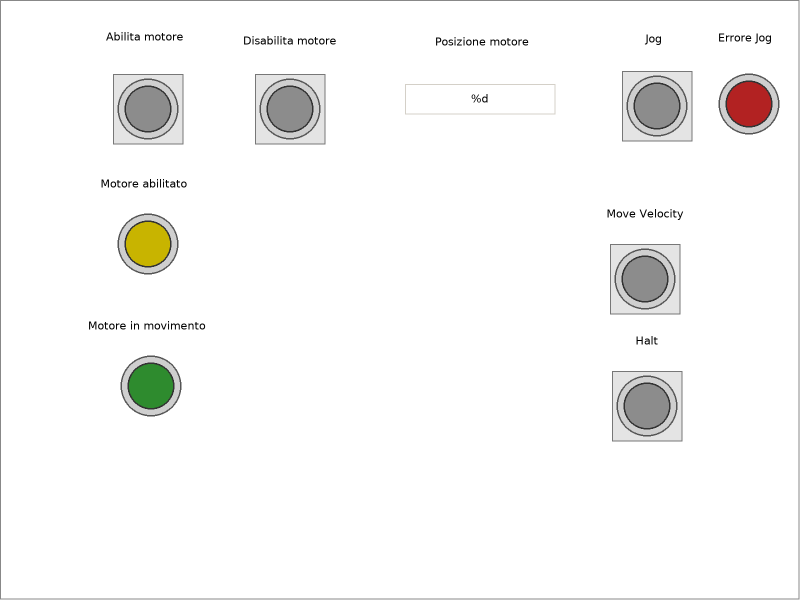
VISUALIZATION Visualization  // 800x600
    PushSwitch (113,74 70x70), variable: GVL.pAbilitaMotore, behaviour: TAP, style: Switch-PushSwitch-Gray
    Lamp1 (113,209 70x70), variable: GVL.motoreAbilitato, style: Lamp-Lamp1-Yellow
    Label (69,169 150x30), "Motore abilitato"
    Label (70,22 150x30), "Abilita motore"
    PushSwitch (255,74 70x70), variable: GVL.pDisabilitaMotore, behaviour: TAP, style: Switch-PushSwitch-Gray
    Label (215,26 150x30), "Disabilita motore"
    Textfield (405,84 150x30), "%d", text variable: GVL.Axis.NcToPlc.ActPos
    PushSwitch (622,71 70x70), variable: GVL.pAbilitaJog, behaviour: TAP, style: Switch-PushSwitch-Gray
    Label (579,24 150x30), "Jog"
    Lamp1 (116,351 70x70), variable: GVL.Axis.Status.Moving, style: Lamp-Lamp1-Green
    Label (72,311 150x30), "Motore in movimento"
    Lamp1 (714,69 70x70), variable: GVL.bErrorJog, style: Lamp-Lamp1-Red
    Label (670,23 150x30), "Errore Jog"
    Label (407,27 150x30), "Posizione motore"
    PushSwitch (610,244 70x70), variable: GVL.pMoveVelocity, behaviour: TAP, style: Switch-PushSwitch-Gray
    Label (570,199 150x30), "Move Velocity"
    PushSwitch (612,371 70x70), variable: GVL.pHalt, behaviour: TAP, style: Switch-PushSwitch-Gray
    Label (572,326 150x30), "Halt"
END_VISUALIZATION

(* stored: Version 1.1.0.1, ProductVersion 3.1.4024.12
   Visu Visualization: Id {f115c04c-1a3c-4c77-b868-9897eb9f7343} *)
